TYPE TcoUrRobotics_O2T_Robot_IO : STRUCT
    bArray AT %Q* : ARRAY[0..23] OF BYTE;
END_STRUCT
END_TYPE

(* stored: Version 1.1.0.1, ProductVersion 3.1.4024.12
   DUT TcoUrRobotics_O2T_Robot_IO: Id {c2ba2317-28e7-0221-0ed3-d9bd1475dc7e} *)
